(* CODESYS project sudoku2.project

Project tree, tasks and I/O mapping:
  Device : CODESYS Control Win V3, 3S - Smart Software Solutions GmbH, order no. 305021, version 3.5.8.10
    application Application
      libraries: Standard, * (System); BASIC, 3.31 (OSCAT); VisuDialogs, * (System)
      task MainTask (cyclic, interval t#20ms, priority 1) calls PLC_PRG
      program PLC_PRG [ST]
      visualisation Visualization
  libraries: VisuSymbols, 3.5.8.0 (System)
  text list GlobalTextList
*)

// Device/Application/PLC_PRG
PROGRAM PLC_PRG
VAR
	square: ARRAY [0..3] OF INT;	(*	Deklaracja tablicy składającej się 
									 	z 4 cyfr typu INT. W programie ta
										tablica zawiera 4 wylosowane numery 
										które reprezentują pola (kwadraty) 
										na planszy. *)
										
	numbers: ARRAY [0..8] OF INT;	(*	Deklaracja tablicy składającej się 
									 	z 9 cyfr typu INT. W programie ta
										tablica zawiera numery w polach
 										na planszy. *)
										
	dis: ARRAY [0..8] OF BOOL;		(*	Deklaracja tablicy składającej się 
									 	z 9 wartości typu BOOL. Jest stworzona 
										bezposrednio aby wylaczac mozliwosc wpisywania 
										do okreslonych pol (deaktywacja). 
										Np dis[5] := TRUE wylacza mozliwosc wpisania 
											do pola 6 (3 kolumna 2 wierz). 
										Uwaga - liczona od 0 *)
										
	good: ARRAY [1..9] OF BOOL;		(*	Deklaracja tablicy składającej się 
									 	z 9 wartości typu BOOL. Jest stworzona 
										do sprawdzania wyniku - zgodnie z zasadami 
										gry sudoku. Np good[2] sprawda czy do planszy 
														wpisano juz cyfre 2. *)
	
	com1: BOOL;		(*	Zmienna reprezentująca pojawienie sie zielonego okna wygranej 
						w wizualizaji *)
					
	com2: BOOL;		//	Zmienna reprezentująca pojawienie sie czerwonego okna  w wizualizaji 

	index: INT;		//	Zmienne wykorzystane do iteracji po pętli FOR 
	index2: INT;	//	(po indeksach tablic zadeklarowanych wyżej)

	war1: BOOL;		(*	Zmienna typu prawda/fałsz, która reprezentuje spełnienie 
						warunku pierwszego do spełnienia aby gracz wygrał. 
						Warunek te odpowiada za to, aby w żadnym polu nie 
						znajdowało się "0" *)
	war2: BOOL;		(*	Zmienna typu prawda/fałsz, która reprezentuje spełnienie 
						warunku pierwszego do spełnienia aby gracz wygrał.
						Warunek te odpowiada za tO, aby w każdym polu 
						znajdowała się unikalna cyfra *)
	
	newGame: BOOL;	//	Zmienna typu prawda/fałsz przypisana do przycisku "nowa gra" w wizualizacji
END_VAR

IF(newGame = TRUE) THEN	
	FOR index:=1 TO 9 BY 1 DO
		good[index] := FALSE;
	END_FOR	

	war1 := FALSE;
	war2 := TRUE;
	
	square[0] := RDM2(low:=0,high:=8,last:=0);
	square[1] := RDM2(low:=0,high:=8,last:=square[0]);
	square[2] := RDM2(low:=0,high:=8,last:=square[1]);
	square[3] := RDM2(low:=0,high:=8,last:=square[2]);
	
	WHILE ((square[0] = square[1]) OR (square[0] = square[2]) OR 
		(square[0] = square[3]) OR (square[1] = square[2]) OR 
		(square[1] = square[3]) OR (square[2] = square[3])) DO
			square[0] := RDM2(low:=0,high:=8,last:=0);
			square[1] := RDM2(low:=0,high:=8,last:=square[0]);
			square[2] := RDM2(low:=0,high:=8,last:=square[1]);
			square[3] := RDM2(low:=0,high:=8,last:=square[2]);
	END_WHILE

	numbers[square[0]] := RDM2(low:=1,high:=9,last:=0);
	numbers[square[1]] := RDM2(low:=1,high:=9,last:=numbers[square[0]]);
	numbers[square[2]] := RDM2(low:=1,high:=9,last:=numbers[square[1]]);
	numbers[square[3]] := RDM2(low:=1,high:=9,last:=numbers[square[2]]);
 
	WHILE ((numbers[square[0]] = numbers[square[1]]) OR (numbers[square[0]] = numbers[square[2]]) OR 
		(numbers[square[0]] = numbers[square[3]]) OR (numbers[square[1]] = numbers[square[2]]) OR 
		(numbers[square[1]] = numbers[square[3]]) OR (numbers[square[2]] = numbers[square[3]])) DO
			numbers[square[0]] := RDM2(low:=1,high:=9,last:=0);
			numbers[square[1]] := RDM2(low:=1,high:=9,last:=numbers[square[0]]);
			numbers[square[2]] := RDM2(low:=1,high:=9,last:=numbers[square[1]]);
			numbers[square[3]] := RDM2(low:=1,high:=9,last:=numbers[square[2]]);
	END_WHILE
	
	FOR index:=0 TO 8 BY 1 DO
		dis[index] := TRUE;
	END_FOR
	
	FOR index:=0 TO 8 BY 1 DO
		IF((index <> square[0]) AND (index <> square[1]) AND 
			(index <> square[2]) AND (index <> square[3])) THEN
				numbers[index] := 0;
				dis[index] := FALSE;
		END_IF
	END_FOR
END_IF

IF((numbers[0]<>0)AND(numbers[1]<>0)AND(numbers[2]<>0)AND(numbers[3]<>0)AND(numbers[4]<>0)
AND(numbers[5]<>0)AND(numbers[6]<>0)AND(numbers[7]<>0)AND(numbers[8]<>0)) THEN
	war1 := TRUE;
END_IF

IF(war1 = TRUE) THEN
	FOR index:=0 TO 8 BY 1 DO
		good[numbers[index]] := TRUE;
	END_FOR
	
	FOR index:=1 TO 9 BY 1 DO
		IF(good[index] = FALSE) THEN
			war2 := FALSE;
			index:=10;
		END_IF
	END_FOR
	
END_IF

IF((war1 = TRUE) AND (war2 = TRUE)) THEN
	com1 := FALSE;
	com2 := TRUE;
	
	dis[0] := TRUE;
	dis[1] := TRUE;
	dis[2] := TRUE;	
	dis[3] := TRUE;	
	dis[4] := TRUE;
	dis[5] := TRUE;
	dis[6] := TRUE;
	dis[7] := TRUE;
	dis[8] := TRUE;
END_IF

IF((war1 = FALSE) OR (war2 = FALSE)) THEN
	com1 := TRUE;
	com2 := FALSE;
END_IF

END_PROGRAM

// Device/Application/Visualization
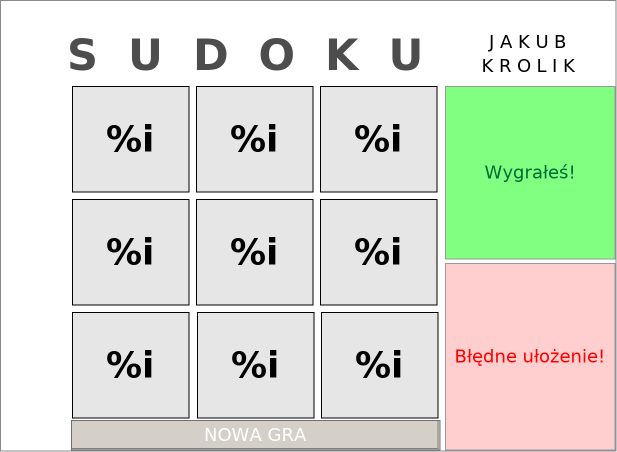
VISUALIZATION Visualization  // 617x452
    Rectangle (72,86 117x106), "%i", text variable: PLC_PRG.numbers[0], input disabled if: PLC_PRG.dis[0]
        OnMouseDown: write PLC_PRG.numbers[0] via Default
    Rectangle (72,199 117x106), "%i", text variable: PLC_PRG.numbers[3], input disabled if: PLC_PRG.dis[3]
        OnMouseDown: write PLC_PRG.numbers[3] via Default
    Rectangle (72,312 117x106), "%i", text variable: PLC_PRG.numbers[6], input disabled if: PLC_PRG.dis[6]
        OnMouseDown: write PLC_PRG.numbers[6] via Default
    Rectangle (196,86 117x106), "%i", text variable: PLC_PRG.numbers[1], input disabled if: PLC_PRG.dis[1]
        OnMouseDown: write PLC_PRG.numbers[1] via Default
    Rectangle (196,199 117x106), "%i", text variable: PLC_PRG.numbers[4], input disabled if: PLC_PRG.dis[4]
        OnMouseDown: write PLC_PRG.numbers[4] via Default
    Rectangle (197,312 117x106), "%i", text variable: PLC_PRG.numbers[7], input disabled if: PLC_PRG.dis[7]
        OnMouseDown: write PLC_PRG.numbers[7] via Default
    Rectangle (320,86 117x106), "%i", text variable: PLC_PRG.numbers[2], input disabled if: PLC_PRG.dis[2]
        OnMouseDown: write PLC_PRG.numbers[2] via Default
    Rectangle (320,199 117x106), "%i", text variable: PLC_PRG.numbers[5], input disabled if: PLC_PRG.dis[5]
        OnMouseDown: write PLC_PRG.numbers[5] via Default
    Rectangle (321,312 117x106), "%i", text variable: PLC_PRG.numbers[8], input disabled if: PLC_PRG.dis[8]
        OnMouseDown: write PLC_PRG.numbers[8] via Default
    Button (71,420 369x30), "NOWA GRA", text variable: PLC_PRG.newGame
        tap PLC_PRG.newGame
    Textfield (445,86 170x173), "Wygrałeś!", invisible if: PLC_PRG.com1
    Textfield (445,263 170x187), "Błędne ułożenie!", invisible if: PLC_PRG.com2
    Label (60,26 371x58), "S U D O K U"
    Label (453,27 150x30), "J A K U B"
    Label (452,51 153x30), "K R O L I K"
END_VISUALIZATION
